TYPE "PositioningMachine_Par"
VERSION : 0.1
// Block: PositioningMachine_Par
   STRUCT
      PosTolerance : LReal;
      DelayInPosition : Time;
      Man : Struct
         VelBwd : LReal;
         VelFwdHigh : LReal;
         VelFwdLow : LReal;
         Acc : LReal;
         Dec : LReal;
         Jerk : LReal;
         DelayChangeVel : Time;
         UsePositionControl : Bool;
      END_STRUCT;
   END_STRUCT;

END_TYPE
